TYPE ST_Identity_PK1_OUT3 :
STRUCT
	ID	:STRING;
	ReadQuality:STRING;
END_STRUCT
END_TYPE

(* stored: Version 1.1.0.1, ProductVersion 3.1.4024.13
   DUT ST_Identity_PK1_OUT3: Id {e162e3cd-2cde-41fe-8180-e99ff98d613d} *)
